# B&R Automation Studio project po_lab2
Automation Studio 4.5.2.102

## Configuration SampleText

### Task classes (Cpu.sw)
```
Cyclic#1 (cycle 2000 us, tolerance 0 us):
  Program <- Program.prg
Binaries: udbdef, TCData, ashwac, arconfig, asfw, ashwd, iomap, User, Role, sysconf
Libraries: sys_lib, Runtime, asstring, DriveLib, McBase
```

### Hardware
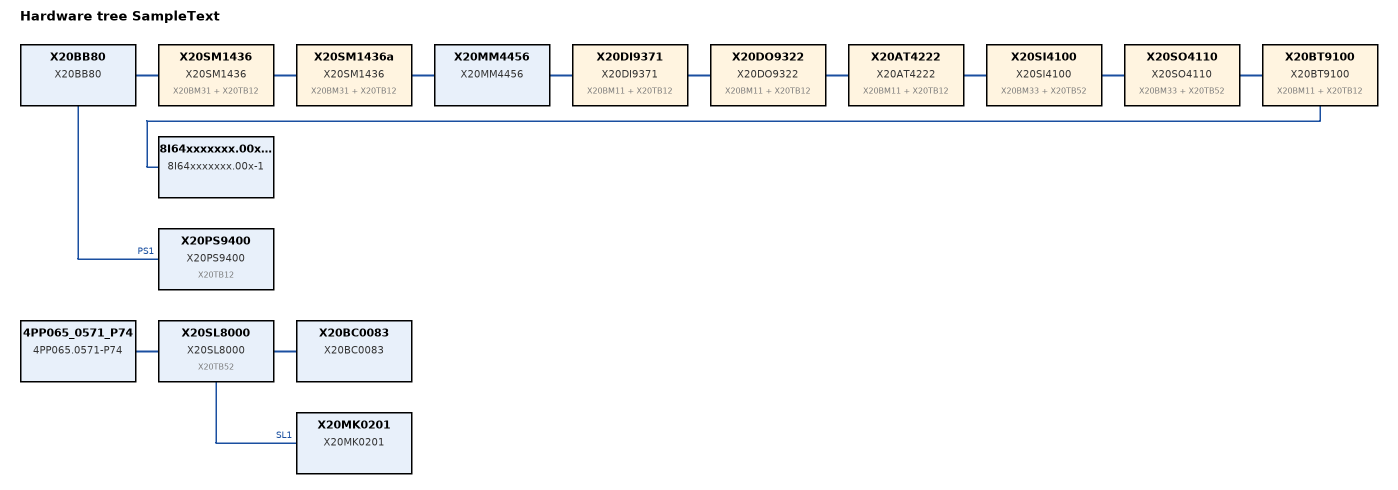
```
4PP065_0571_P74 : 4PP065.0571-P74 v1.1.2.0
  Connector IF4:
    EplInterfaceRedundant = 0
    EplEthInterfaceRedundant = 0
  Connector IF5:
    ActivateDevice = 1
    Mode = Manual
    InternetAddress = 10.0.1.10
    SubnetMask = 255.255.255.0
  ConfigurationID = labBR
  Simulation = 1
  TimerDeviceType = EPLX2X
  TimerDevice = 4PP065_0571_P74.IF4
  TaskClassIdleTime = 2000
  Cyclic1Duration = 2000
  Cyclic1Tolerance = 0
  Cyclic1Output = 1
8I64xxxxxxx.00x-1 : 8I64xxxxxxx.00x-1 v1.3.9.1  [X2X1 -> X20BT9100.X2X1 [Cable Type=X2XCable, Length=10, Version=1.0.0.2]]
  FunctionModel = Standard
  packedETAD = packed
  packedETI = packed
  packedCMDD = packed
  packedCMI = packed
  UNS = 220
  NCR = 10
  NSP = 890
  COS = 64
  RSC = 33000
X20AT4222 : X20AT4222 v1.2.3.0  [SS1 -> X20TB12e.SS; SL -> X20BM11c.SL1]
X20BB80 : X20BB80 v1.0.2.0
X20BC0083 : X20BC0083 v2.9.0.0  [PLK1 -> X20SL8000.PLK2 (NodeNumber=2) [Cable Type=PowerlinkCable, Length=10, Version=1.0.0.2]; SL -> X20BB80.SL1]
X20BM11 : X20BM11 v1.0.0.1  [X2X1 -> X20BM33a.X2X2]
X20BM11a : X20BM11 v1.0.0.1  [X2X1 -> X20MM4456.X2X2]
X20BM11b : X20BM11 v1.0.0.1  [X2X1 -> X20BM11a.X2X2]
X20BM11c : X20BM11 v1.0.0.1  [X2X1 -> X20BM11b.X2X2]
X20BM31 : X20BM31 v1.0.0.1  [X2X1 -> X20BB80.IF1]
X20BM31a : X20BM31 v1.0.0.1  [X2X1 -> X20BM31.X2X2]
X20BM33 : X20BM33 v1.0.0.4  [X2X1 -> X20BM11c.X2X2]
X20BM33a : X20BM33 v1.0.0.4  [X2X1 -> X20BM33.X2X2]
X20BT9100 : X20BT9100 v1.0.3.0  [SS1 -> X20TB12f.SS; SL -> X20BM11.SL1]
X20DI9371 : X20DI9371 v1.0.2.0  [SS1 -> X20TB12c.SS; SL -> X20BM11a.SL1]
X20DO9322 : X20DO9322 v1.0.3.0  [SS1 -> X20TB12d.SS; SL -> X20BM11b.SL1]
X20MK0201 : X20MK0201 v1.0.0.0  [SL -> X20SL8000.SL1]
X20MM4456 : X20MM4456 v1.1.5.0  [X2X1 -> X20BM31a.X2X2]
X20PS9400 : X20PS9400 v1.0.2.4  [SS1 -> X20TB12.SS; PS -> X20BB80.PS1]
X20SI4100 : X20SI4100 v1.10.1.1  [SS1 -> X20TB52.SS; SL -> X20BM33.SL1]
X20SL8000 : X20SL8000 v1.6.5.1  [PLK1 -> 4PP065_0571_P74.IF4 [Cable Type=PowerlinkCable, Length=10, Version=1.0.0.2]; PLK2 -> X20BC0083.PLK1 [Cable Type=PowerlinkCable, Length=10, Version=1.0.0.2]; SS1 -> X20TB52b.SS]
  SafeProject = SafeLOGIC-1
  SafeDesigner = 3.0.18.3402403
X20SM1436 : X20SM1436 v2.2.0.0  [SS1 -> X20TB12a.SS; SL -> X20BM31.SL1]
X20SM1436a : X20SM1436 v2.2.0.0  [SS1 -> X20TB12b.SS; SL -> X20BM31a.SL1]
X20SO4110 : X20SO4110 v1.10.1.1  [SS1 -> X20TB52a.SS; SL -> X20BM33a.SL1]
  SafeModuleID = 3
X20TB12 : X20TB12 v1.0.0.0
X20TB12a : X20TB12 v1.0.0.0
X20TB12b : X20TB12 v1.0.0.0
X20TB12c : X20TB12 v1.0.0.0
X20TB12d : X20TB12 v1.0.0.0
X20TB12e : X20TB12 v1.0.0.0
X20TB12f : X20TB12 v1.0.0.0
X20TB52 : X20TB52 v1.0.0.1
X20TB52a : X20TB52 v1.0.0.1
X20TB52b : X20TB52 v1.0.0.1
```

### IoMap.iom - 4PP065_0571_P74/IoMap.iom
```iecst
VAR_CONFIG
	::Program:driveSM.state AT %IW."8I64xxxxxxx.00x-1".ETAD_Input;
	::Program:driveSM.command AT %QW."8I64xxxxxxx.00x-1".CMDD_Output;
	::Program:driveSM.speed AT %QW."8I64xxxxxxx.00x-1".LFRD_Output;
	::Program:doorSM.direction AT %IX."X20DI9371".DigitalInput01;
	::Program:doorSM.sw1 AT %IX."X20DI9371".DigitalInput02;
	::Program:doorSM.sw2 AT %IX."X20DI9371".DigitalInput03;
	::Program:doorSM.sw3 AT %IX."X20DI9371".DigitalInput04;
	::Program:doorSM.sw4 AT %IX."X20DI9371".DigitalInput05;
	::Program:ledSM.led1 AT %QX."X20DO9322".DigitalOutput02;
	::Program:ledSM.led2 AT %QX."X20DO9322".DigitalOutput03;
	::Program:ledSM.led3 AT %QX."X20DO9322".DigitalOutput04;
	::Program:ledSM.led4 AT %QX."X20DO9322".DigitalOutput05;
END_VAR
```

## Logical view

Binary libraries used (declarations not repeated): Runtime, Operator, AsIecCon, astime, sys_lib, asstring, McBase

### Library Logical/Libraries/DriveLib (ANSIC)

#### Types.typ
```iecst
TYPE
	DoorStates :
		(
		ST_INIT, (*Initialization of parameters and waiting for switching on of frequency converter*)
		ST_UNKNOWN, (*Gates are in unknown state*)
		ST_OPEN, (*Gates are opened*)
		ST_CLOSE, (*Gates are closed*)
		ST_ACC_POS, (*Acceleration of gates torwards opening*)
		ST_ACC_NEG, (*Acceleration of gates torwards closing*)
		ST_POS, (*Moving torwards opening *)
		ST_NEG, (*Moving torwards closing*)
		ST_DEC_POS, (*Slowing torwards opening*)
		ST_DEC_NEG (*Slowing torwards closing*)
		);
	EtadCodes :
		(
		STATE_DISABLED := 64,
		CMD_SWITCHED_ON := 35,
		STATE_READY := 33
		);
	CmddCodes :
		(
		CMD_SHUTDOWN := 6,
		STATE_SWITCHED_ON := 7,
		CMD_ENABLED := 15
		);
END_TYPE
```

#### DriveLib.fun
```iecst
{REDUND_ERROR} FUNCTION_BLOCK DriveStateMachine (*TODO: Add your comment here*) (*$GROUP=User,$CAT=User,$GROUPICON=User.png,$CATICON=User.png*)
	VAR_INPUT
		state : {REDUND_UNREPLICABLE} UINT; (*State of frequency converter*)
		enable : {REDUND_UNREPLICABLE} BOOL; (*Work signal for FB*)
	END_VAR
	VAR_OUTPUT
		command : {REDUND_UNREPLICABLE} UINT; (*Command to frequency converter*)
		speed : {REDUND_UNREPLICABLE} INT; (*Set speed*)
	END_VAR
END_FUNCTION_BLOCK

{REDUND_ERROR} FUNCTION_BLOCK DoorStateMachine (*TODO: Add your comment here*) (*$GROUP=User,$CAT=User,$GROUPICON=User.png,$CATICON=User.png*)
	VAR_INPUT
		state : UINT; (*State of frequency converter*)
		direction : {REDUND_UNREPLICABLE} BOOL; (*Command to frequency converter*)
		sw4 : {REDUND_UNREPLICABLE} BOOL; (*Signal of end-switch4*)
		sw3 : {REDUND_UNREPLICABLE} BOOL; (*Signal of end-switch3*)
		sw2 : {REDUND_UNREPLICABLE} BOOL; (*Signal of end-switch2*)
		sw1 : {REDUND_UNREPLICABLE} BOOL; (*Signal of end-switch1*)
	END_VAR
	VAR_OUTPUT
		speed : {REDUND_UNREPLICABLE} INT; (*Set speed*)
	END_VAR
END_FUNCTION_BLOCK

{REDUND_ERROR} {REDUND_UNREPLICABLE} FUNCTION_BLOCK LedStateMachine (*TODO: Add your comment here*) (*$GROUP=User,$CAT=User,$GROUPICON=User.png,$CATICON=User.png*)
	VAR_INPUT
		state : {REDUND_UNREPLICABLE} UINT; (*State of frequency converter*)
	END_VAR
	VAR_OUTPUT
		led1 : {REDUND_UNREPLICABLE} BOOL; (*Work signal of frequency converter*)
		led2 : {REDUND_UNREPLICABLE} BOOL; (*Work signal of frequency converter*)
		led3 : {REDUND_UNREPLICABLE} BOOL; (*Work signal of frequency converter*)
		led4 : {REDUND_UNREPLICABLE} BOOL; (*Work signal of frequency converter*)
		timer : {REDUND_UNREPLICABLE} INT; (*Set speed*)
	END_VAR
END_FUNCTION_BLOCK
```

#### DoorStateMachine.c
```c
#include <bur/plctypes.h>
#ifdef __cplusplus
	extern "C"
	{
#endif
	#include "DriveLib.h"
#ifdef __cplusplus
	};
#endif
/* TODO: Add your comment here */
void DoorStateMachine(struct DoorStateMachine* inst)
{
	/*TODO: Add your code here*/
	switch(inst->state){
		case ST_INIT:
			{
				if(inst->sw1==0 && inst->sw2==0 && inst->sw3==0 && inst->sw4==0)
					inst->state=ST_UNKNOWN;
				break;
			}

		case ST_UNKNOWN:
			{
				if(inst->direction == 1 && inst->sw4 == 1)
					inst->state = ST_CLOSE;
				if(inst->direction == 0 && inst->sw1 == 0)
					inst->state = ST_OPEN;

			}

		case ST_CLOSE:
			{
				inst->speed = 0;
				if(inst->direction==1 && inst->sw4 == 0)
					inst->state=ST_ACC_POS;
				break;
			}
		case ST_ACC_POS:
			{
				inst->speed = 800;
				if(inst->direction==1 && inst->sw3 == 0)
					inst->state=ST_POS;
				if(inst->direction==0)
					inst->state=ST_DEC_NEG;
				break;
			}

		case ST_POS:
			{
				inst->speed = 450;
				if(inst->direction==1 && inst->sw2==0)
					inst->state=ST_DEC_POS;
				if(inst->direction==0)
					inst->state=ST_NEG;
				break;
			}
		case ST_DEC_POS:
			{
				inst->speed = 150;
				if(inst->direction==1 && inst->sw1 == 0)
					inst->state=ST_OPEN;

				break;
			}
		case ST_OPEN:
			{
				inst->speed = 0;
				if(inst->direction==0 && inst->sw1==1)
					inst->state=ST_ACC_NEG;
				break;
			}

		case ST_ACC_NEG:
			{
				inst->speed = -800;
				if(inst->direction==0 && inst->sw2==1 )
					inst->state=ST_NEG;
				if(inst->direction==1)
					inst->state=ST_DEC_POS;
				break;
			}
		case ST_NEG:
			{
				inst->speed = -450;
				if(inst->direction==0 && inst->sw3==1)
					inst->state=ST_DEC_NEG;
				if(inst->direction==1)
					inst->state=ST_POS;
				break;

			}
		case ST_DEC_NEG:
			{
				inst->speed = -150;
				if(inst->direction==0 && inst->sw4 == 1)
					inst->state=ST_CLOSE;
				break;
			}
	}
}
```

#### LedStateMachine.c
```c
#include <bur/plctypes.h>
#ifdef __cplusplus
	extern "C"
	{
#endif
	#include "DriveLib.h"
#ifdef __cplusplus
	};
#endif
/* TODO: Add your comment here */
void LedStateMachine(struct LedStateMachine* inst)
{
	switch(inst->state)
	{
		case ST_INIT:
			{
				inst->led1=0;
				inst->led2=0;
				inst->led3=0;
				inst->led4=0;
				break;
			}

		case ST_UNKNOWN:
			{
				if(inst->timer%11==10)
				{
					inst->led1=!inst->led1;
					inst->led2=!inst->led2;
					inst->led3=!inst->led3;
					inst->led4=!inst->led4;
				}
				break;
			}

		case ST_CLOSE:
			{
				inst->led1=1;
				inst->led2=1;
				inst->led3=1;
				inst->led4=1;
				break;
			}
		case ST_ACC_POS:
			{
				inst->led1=1;
				inst->led2=1;
				inst->led3=1;
				if(inst->timer%11==10)
					inst->led4=!inst->led4;
				break;
			}
		case ST_POS:
			{
				inst->led1=1;
				inst->led2=1;
				if(inst->timer%21==20)
					inst->led3=!inst->led3;
				inst->led4=0;
				break;
			}
		case ST_DEC_POS:
			{
				inst->led1=1;
				if(inst->timer%21==20)
					inst->led2=!inst->led2;
				inst->led3=0;
				inst->led4=0;
				break;
			}

		case ST_OPEN:
			{
				inst->led1=0;
				inst->led2=0;
				inst->led3=0;
				inst->led4=0;
				break;
			}

		case ST_ACC_NEG:
			{
				if(inst->timer%11==10)
					inst->led1=!inst->led1;
				inst->led2=0;
				inst->led3=0;
				inst->led4=0;
				break;
			}
		case ST_NEG:
			{
				inst->led1=1;
				if(inst->timer%21==20)
					inst->led2=!inst->led2;
				inst->led3=0;
				inst->led4=0;
				break;
			}

		case ST_DEC_NEG:
			{
				inst->led1=1;
				inst->led2=1;
				if(inst->timer%21==20)
					inst->led3=!inst->led3;
				inst->led4=0;
				break;

			}
	}
	inst->timer++;
}
```

### Program Logical/Program

#### Variables.var
```iecst
VAR
	ledSM : LedStateMachine := (0);
	driveSM : DriveStateMachine := (0);
	doorSM : DoorStateMachine := (0);
END_VAR
```

#### Init.c
```c
#include <bur/plctypes.h>

#ifdef _DEFAULT_INCLUDES
	#include <AsDefault.h>
#endif

void _INIT ProgramInit(void)
{
	driveSM.enable = 1;
	driveSM.speed = 50;
}
```
